FUNCTION_BLOCK FB_DataChannelRecvFifo EXTENDS FB_ArrayFifo
VAR_INPUT
END_VAR
VAR_OUTPUT
END_VAR
VAR
	m_pDataChannel				: POINTER TO FB_DataChannelRecvBase;
	m_bolEnable					: BOOL;
	m_intMaxFifoSize			: INT  := 10;
	m_pItem						: POINTER TO BYTE;
	m_bolResult					: BOOL;
END_VAR

IF m_bolEnable AND (m_pItem <> Tc3_MemMan.NULL) THEN
	IF NOT m_pDataChannel^.Busy THEN
		m_bolResult := m_pDataChannel^.GetData(
						udiDataSize := m_pDataChannel^.DataSize,
						pData		:= m_pItem);

		IF m_uinItemCount < m_uinMaxItemCount THEN
			Push(m_pItem);
		ELSE
			m_pDataChannel^.Error := 1;
		END_IF 	
	END_IF
	
	m_pDataChannel^();
END_IF

PROPERTY PUBLIC Item : POINTER TO BYTE
SET
m_pItem := Item;
END_SET
GET
END_GET
END_PROPERTY

PROPERTY PUBLIC Enable : BOOL
SET
m_bolEnable := Enable;
END_SET
GET
Enable := m_bolEnable;
END_GET
END_PROPERTY

PROPERTY PUBLIC DataChannel : POINTER TO FB_DataChannelRecvBase
SET
m_pDataChannel := DataChannel;
END_SET
END_PROPERTY

PROPERTY PUBLIC MaxFifoSize : INT
GET
MaxFifoSize := m_intMaxFifoSize;
END_GET
SET
m_intMaxFifoSize := MaxFifoSize;
END_SET
END_PROPERTY

END_FUNCTION_BLOCK

(* stored: Version 1.1.0.1, ProductVersion 3.1.0.24
   POU FB_DataChannelRecvFifo: Id {ae597d08-4a69-42c6-9fb0-3008c460e2f1}
   Property Item: Id {62be58f2-7569-483b-a49f-67f61f58529e}
   Set Set: Id {3aee014a-e624-441d-9a5f-55fee3fac0ed}
   Get Get: Id {8bc4f753-0ac8-495e-896b-f1318ba9c596}
   Property Enable: Id {63bf5842-61e2-488d-97c1-116ec3d2f9bc}
   Set Set: Id {1ea626ac-b4fe-4b96-9184-00277b85e001}
   Get Get: Id {c1f3703b-41a7-4ced-a19a-4e16cb6e446c}
   Property DataChannel: Id {913bfa4f-e7e4-439a-98b8-7080b88d78ea}
   Set Set: Id {5c04e000-f701-402a-b897-0e080306905c}
   Property MaxFifoSize: Id {a599e5e1-d0cb-49f1-af78-ed1ab3faac08}
   Get Get: Id {bd85c2b6-85dd-4032-9f5a-21525ea64c92}
   Set Set: Id {f3c4eafc-a7cd-4917-9e2a-e683c3ac73c2} *)
